FUNCTION_BLOCK REC_Queue
VAR_INPUT
END_VAR
VAR_OUTPUT
END_VAR
VAR
END_VAR

METHOD Count_Queue
VAR_INPUT
END_VAR
END_METHOD

METHOD Delete_Queue
VAR_INPUT
END_VAR
END_METHOD

METHOD Empty_Queue
VAR_INPUT
END_VAR
END_METHOD

METHOD Full_Queue
VAR_INPUT
END_VAR
END_METHOD

METHOD Head_Queue
VAR_INPUT
END_VAR
END_METHOD

METHOD Init_Queue
VAR_INPUT
END_VAR
END_METHOD

METHOD Insert_Queue
VAR_INPUT
END_VAR
END_METHOD

END_FUNCTION_BLOCK

(* stored: Version 1.1.0.1, ProductVersion 3.1.4018.5
   POU REC_Queue: Id {832394c0-1517-48e2-8c89-b76fea609dd7}, SpecialFunc None
   Method Count_Queue: Id {686262fd-2396-4462-81b8-5b181d3f2c6f}
   Method Delete_Queue: Id {55ded70a-c88b-47b8-bb22-6533aafbb848}
   Method Empty_Queue: Id {4a105195-4dd5-475c-bf44-a3e7dc5552da}
   Method Full_Queue: Id {5cec573b-8d8a-436c-9c16-db07a6ea5440}
   Method Head_Queue: Id {fd96c293-b0fd-47cf-8959-99c3b5a08f6b}
   Method Init_Queue: Id {e62adc94-f1a3-4959-86d8-40a71887af54}
   Method Insert_Queue: Id {82e0b24e-c50c-4ed1-a77e-80a5926b03f4} *)
